PROGRAM MAIN
VAR
END_VAR

END_PROGRAM

(* stored: Version 1.1.0.1
   POU MAIN: Id {21979fe2-12a4-4c59-bbdc-5afb35665cf8} *)
